# EPICS IOC start-up script: iocsh/julabof25hl.iocsh
dbLoadRecords(JULABOF25HL.db, "P=$(P), PORT=$(PORT), ADDR=$(ADDR), TEMPSCAN=$(TEMPSCAN), SETPNAME=$(SETPNAME), SETPNR=$(SETPNR)")
